//{attribute 'qualified_only'}
//{attribute 'strict'}
{attribute 'to_string'}
{attribute 'to_wstring'}
TYPE E_M001_Settings :
(
	//eSt001_Settings_none := 0,
	
	eM001_Settings_Deaktiv,		// Station deaktivieren
	eM001_Settings_Autohome,	// automatic home with start button
	
	//eM001_Settings_PalletLayout,	// Palettenlayout (1-4)
	
	/// has to be set to last index for array bounds!
	eM001_Settings_nMaxIdx	
);
END_TYPE

(* stored: Version 1.1.0.1
   DUT E_M001_Settings: Id {ef593c5c-4671-414f-b686-79ac0bbb7160} *)
